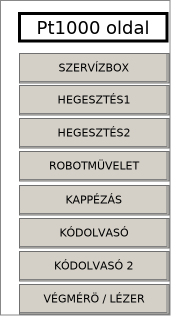
VISUALIZATION Tengely_Pt1000_beallitasok  // 171x316
    RoundedRectangle (18,12 150x30)
    Label (18,13 150x30), "Pt1000 oldal"
    Button (19,118 150x30), "HEGESZTÉS2"
        OnMouseUp: execute { GVL.iFoLapozo:=GVL.SZERVIZ_FUL; GVL.iSzervizLapozo:=GVL.HEGESZTES_FUL; }
    Button (19,53 150x30), "SZERVÍZBOX"
        OnMouseUp: execute {
            GVL.iFoLapozo:=GVL.SZERVIZ_FUL;
            GVL.iSzervizLapozo:=GVL.BEHELYEZES_FUL;
            GVL.iTengelyLapozo:=GVL.PT_TENGELY_FUL;
        }
    Button (19,85 150x30), "HEGESZTÉS1"
        OnMouseUp: execute { GVL.iFoLapozo:=GVL.SZERVIZ_FUL; GVL.iSzervizLapozo:=GVL.HEGESZTES_FUL; }
    Button (19,151 150x30), "ROBOTMÜVELET"
        OnMouseUp: execute { GVL.iFoLapozo:=GVL.SZERVIZ_FUL; GVL.iSzervizLapozo:=GVL.ROBOT_FUL; }
    Button (19,284 150x30), "VÉGMÉRÖ / LÉZER"
        OnMouseUp: execute { GVL.iFoLapozo:=GVL.SZERVIZ_FUL; GVL.iSzervizLapozo:=GVL.VEGMERO_FUL; }
    Button (19,185 150x30), "KAPPÉZÁS"
        OnMouseUp: execute { GVL.iFoLapozo:=GVL.SZERVIZ_FUL; GVL.iSzervizLapozo:=GVL.KAPPE_PRES_FUL; }
    Button (19,218 150x30), "KÓDOLVASÓ"
        OnMouseUp: execute { GVL.iFoLapozo:=GVL.SZERVIZ_FUL; GVL.iSzervizLapozo:=GVL.KODOLVASO_FUL; }
    Button (19,251 150x30), "KÓDOLVASÓ 2"
        OnMouseUp: execute { GVL.iFoLapozo:=GVL.SZERVIZ_FUL; GVL.iSzervizLapozo:=GVL.KODOLVASO_FUL; }
END_VISUALIZATION

(* stored: Version 1.1.0.1, ProductVersion 3.1.4024.11
   Visu Tengely_Pt1000_beallitasok: Id {933d92fb-815e-4a61-9e06-825a4e5b330a} *)
